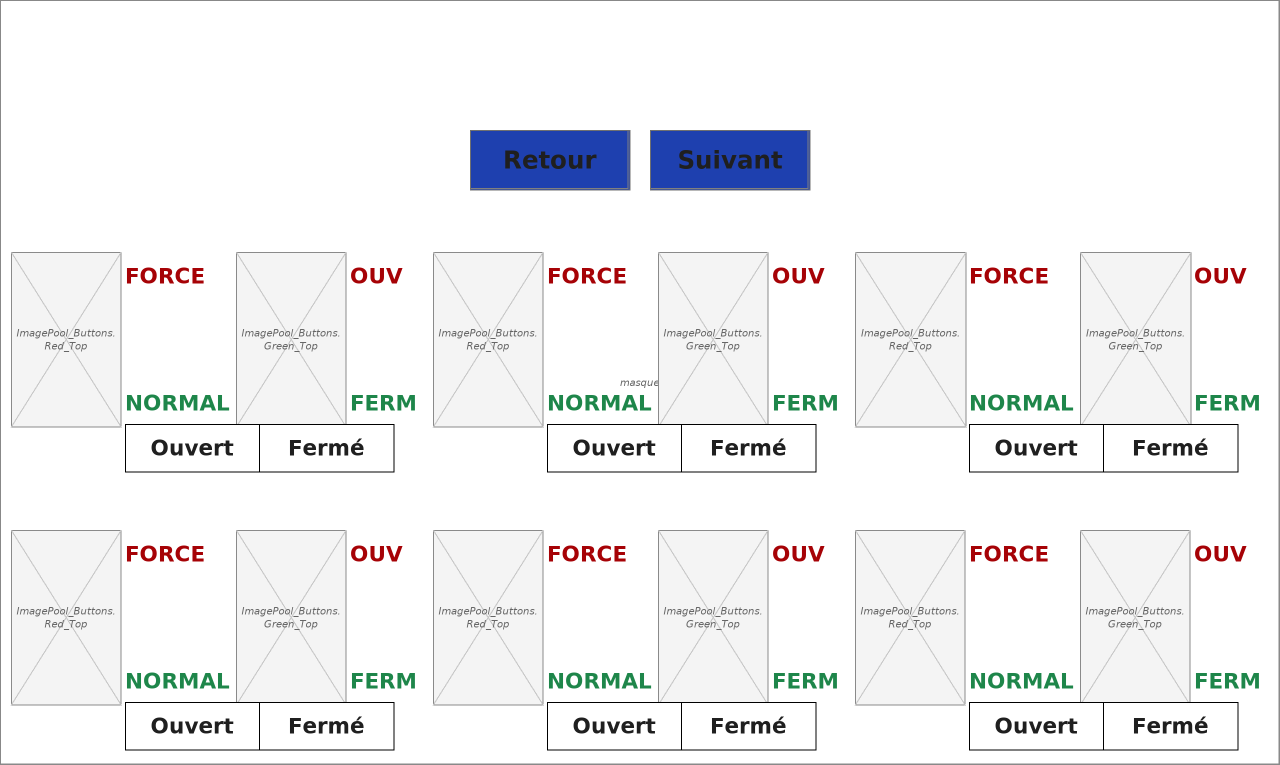
VISUALIZATION Maintenance_2  // 1280x765
    Frame (0,0 1280x765)
        shows masque()
    Button (650,130 160x60), "Suivant"
        OnMouseDown: execute {
            IF (Option_Bas_Debit OR Option_Douchette OR Option_NEP)
            	THEN
            	VisuElems.CURRENTVISU := 'Maintenance_3';
            	ELSIF (Option_WC_GV OR Option_WC_PV OR Option_Prise)
            		THEN
            		VisuElems.CURRENTVISU := 'Maintenance_4';
            	ELSIF (Option_Cabine_Climatique)
            		THEN
            		VisuElems.CURRENTVISU := 'Maintenance_5';
            	ELSIF (Option_Com_RegSouf_Ultrason)
            		THEN
            		VisuElems.CURRENTVISU := 'Maintenance_6';
            	ELSE
            		VisuElems.CURRENTVISU := 'Maintenance_7';
            END_IF
        }
    Button (470,130 160x60), "Retour"
        OnMouseDown: execute {
            IF (Option_RegSouf_Ultrason OR Option_Reg_Etanche_Ext OR Option_V3V_EauMitig)
            	THEN
            	VisuElems.CURRENTVISU := 'Maintenance_1';
            	ELSE
            	VisuElems.CURRENTVISU := 'menu';
            END_IF
        }
    Group (433,212 415x260), invisible if: NOT Option_Douche OR Option_Debitmetre_Douche
        Group (0,40 415x174)
            Group (0,0 225x175)
                Group (0,0 110x175)
                    Image (0,0 110x175), invisible if: EF_Cmd_Vanne_Alim_Douche, image: ImagePool_Buttons.Green_Bottom
                        OnMouseDown: toggle EF_Cmd_Vanne_Alim_Douche
                    Image (0,0 110x175), invisible if: NOT EF_Cmd_Vanne_Alim_Douche, image: ImagePool_Buttons.Red_Top
                        OnMouseDown: toggle EF_Cmd_Vanne_Alim_Douche
                Rectangle (111,0 114x48), "FORCE"
                Rectangle (111,64 114x48), "MODE"
                Rectangle (111,127 114x48), "NORMAL"
            Group (225,0 190x175), invisible if: NOT EF_Cmd_Vanne_Alim_Douche
                Group (0,0 110x175)
                    Image (0,0 110x175), invisible if: F_Cmd_Vanne_Alim_Douche, image: ImagePool_Buttons.Red_Bottom
                        OnMouseDown: toggle F_Cmd_Vanne_Alim_Douche
                    Image (0,0 110x175), invisible if: NOT F_Cmd_Vanne_Alim_Douche, image: ImagePool_Buttons.Green_Top
                        OnMouseDown: toggle F_Cmd_Vanne_Alim_Douche
                Rectangle (111,0 79x48), "OUV"
                Rectangle (111,64 79x48), "OUT"
                Rectangle (111,127 79x48), "FERM"
        Group (33,212 350x48)
            Rectangle (0,0 81x48), "FDC :"
            RoundedRectangle (81,0 135x48), "Ouvert", invisible if: NOT E_Vanne_Alim_Douche_Ouv
            RoundedRectangle (215,0 135x48), "Fermé", invisible if: NOT E_Vanne_Alim_Douche_Ferm
        Rectangle (0,0 415x40), "Vanne douche"
    Group (433,490 415x260), invisible if: NOT Option_Lavabo OR Option_Debitmetre_Lavabo
        Group (0,40 415x174)
            Group (0,0 225x175)
                Group (0,0 110x175)
                    Image (0,0 110x175), invisible if: EF_Cmd_Vanne_Alim_Douche, image: ImagePool_Buttons.Green_Bottom
                        OnMouseDown: toggle EF_Cmd_Vanne_Alim_Douche
                    Image (0,0 110x175), invisible if: NOT EF_Cmd_Vanne_Alim_Douche, image: ImagePool_Buttons.Red_Top
                        OnMouseDown: toggle EF_Cmd_Vanne_Alim_Douche
                Rectangle (111,0 114x48), "FORCE"
                Rectangle (111,64 114x48), "MODE"
                Rectangle (111,127 114x48), "NORMAL"
            Group (225,0 190x175), invisible if: NOT EF_Cmd_Vanne_Alim_Douche
                Group (0,0 110x175)
                    Image (0,0 110x175), invisible if: F_Cmd_Vanne_Alim_Douche, image: ImagePool_Buttons.Red_Bottom
                        OnMouseDown: toggle F_Cmd_Vanne_Alim_Douche
                    Image (0,0 110x175), invisible if: NOT F_Cmd_Vanne_Alim_Douche, image: ImagePool_Buttons.Green_Top
                        OnMouseDown: toggle F_Cmd_Vanne_Alim_Douche
                Rectangle (111,0 79x48), "OUV"
                Rectangle (111,64 79x48), "OUT"
                Rectangle (111,127 79x48), "FERM"
        Group (33,212 350x48)
            Rectangle (0,0 81x48), "FDC :"
            RoundedRectangle (81,0 135x48), "Ouvert", invisible if: NOT E_Vanne_Alim_Lavabo_Ouv
            RoundedRectangle (215,0 135x48), "Fermé", invisible if: NOT E_Vanne_Alim_Lavabo_Ferm
        Rectangle (0,0 415x40), "Vanne lavabo"
    Group (855,212 415x260), invisible if: NOT Option_Douche
        Group (0,40 415x174)
            Group (0,0 225x175)
                Group (0,0 110x175)
                    Image (0,0 111x175), invisible if: EF_Cmd_Vanne_Vid_Douche, image: ImagePool_Buttons.Green_Bottom
                        OnMouseDown: toggle EF_Cmd_Vanne_Vid_Douche
                    Image (0,0 111x175), invisible if: NOT EF_Cmd_Vanne_Vid_Douche, image: ImagePool_Buttons.Red_Top
                        OnMouseDown: toggle EF_Cmd_Vanne_Vid_Douche
                Rectangle (111,0 114x48), "FORCE"
                Rectangle (111,64 114x48), "MODE"
                Rectangle (111,127 114x48), "NORMAL"
            Group (225,0 190x175), invisible if: NOT EF_Cmd_Vanne_Vid_Douche
                Group (0,0 110x175)
                    Image (0,0 111x175), invisible if: F_Cmd_Vanne_Vid_Douche, image: ImagePool_Buttons.Red_Bottom
                        OnMouseDown: toggle F_Cmd_Vanne_Vid_Douche
                    Image (0,0 111x175), invisible if: NOT F_Cmd_Vanne_Vid_Douche, image: ImagePool_Buttons.Green_Top
                        OnMouseDown: toggle F_Cmd_Vanne_Vid_Douche
                Rectangle (111,0 79x48), "OUV"
                Rectangle (111,64 79x48), "OUT"
                Rectangle (111,127 79x48), "FERM"
        Group (33,212 350x48)
            Rectangle (0,0 81x48), "FDC :"
            RoundedRectangle (81,0 135x48), "Ouvert", invisible if: NOT E_Vanne_Vidange_Douche_Ouv
            RoundedRectangle (215,0 135x48), "Fermé", invisible if: NOT E_Vanne_Vidange_Douche_Ferm
        Rectangle (0,0 415x40), "Drain douche"
    Group (855,490 415x260), invisible if: NOT Option_Lavabo
        Group (0,40 415x174)
            Group (0,0 225x175)
                Group (0,0 110x175)
                    Image (0,0 110x175), invisible if: EF_Cmd_Vanne_Vid_Lavabo, image: ImagePool_Buttons.Green_Bottom
                        OnMouseDown: toggle EF_Cmd_Vanne_Vid_Lavabo
                    Image (0,0 110x175), invisible if: NOT EF_Cmd_Vanne_Vid_Lavabo, image: ImagePool_Buttons.Red_Top
                        OnMouseDown: toggle EF_Cmd_Vanne_Vid_Lavabo
                Rectangle (111,0 114x48), "FORCE"
                Rectangle (111,64 114x48), "MODE"
                Rectangle (111,127 114x48), "NORMAL"
            Group (225,0 190x175), invisible if: NOT EF_Cmd_Vanne_Vid_Lavabo
                Group (0,0 110x175)
                    Image (0,0 110x175), invisible if: F_Cmd_Vanne_Vid_Lavabo, image: ImagePool_Buttons.Red_Bottom
                        OnMouseDown: toggle F_Cmd_Vanne_Vid_Lavabo
                    Image (0,0 110x175), invisible if: NOT F_Cmd_Vanne_Vid_Lavabo, image: ImagePool_Buttons.Green_Top
                        OnMouseDown: toggle F_Cmd_Vanne_Vid_Lavabo
                Rectangle (111,0 79x48), "OUV"
                Rectangle (111,64 79x48), "OUT"
                Rectangle (111,127 79x48), "FERM"
        Group (33,212 350x48)
            Rectangle (0,0 81x48), "FDC :"
            RoundedRectangle (81,0 135x48), "Ouvert", invisible if: NOT E_Vanne_Vidange_Lavabo_Ouv
            RoundedRectangle (215,0 135x48), "Fermé", invisible if: NOT E_Vanne_Vidange_Lavabo_Ferm
        Rectangle (0,0 415x40), "Drain lavabo"
    Group (11,212 415x260), invisible if: NOT Option_Douche OR NOT Option_Debitmetre_Douche
        Group (0,40 415x174)
            Group (0,0 225x175)
                Group (0,0 110x175)
                    Image (0,0 110x175), invisible if: EF_Cmd_ElectroValve_Alim_Douche, image: ImagePool_Buttons.Green_Bottom
                    Image (0,0 110x175), invisible if: NOT EF_Cmd_ElectroValve_Alim_Douche, image: ImagePool_Buttons.Red_Top
                Rectangle (111,0 114x48), "FORCE"
                Rectangle (111,64 114x48), "MODE"
                Rectangle (111,127 114x48), "NORMAL"
            Group (225,0 190x175), invisible if: NOT EF_Cmd_ElectroValve_Alim_Douche
                Group (0,0 110x175)
                    Image (0,0 110x175), invisible if: F_Cmd_ElectroValve_Alim_Douche, image: ImagePool_Buttons.Red_Bottom
                        OnMouseDown: toggle F_Cmd_ElectroValve_Alim_Douche
                    Image (0,0 110x175), invisible if: NOT F_Cmd_ElectroValve_Alim_Douche, image: ImagePool_Buttons.Green_Top
                        OnMouseDown: toggle F_Cmd_ElectroValve_Alim_Douche
                Rectangle (111,0 79x48), "OUV"
                Rectangle (111,64 79x48), "OUT"
                Rectangle (111,127 79x48), "FERM"
        Group (33,212 350x48), invisible if: TRUE
            Rectangle (0,0 81x48), "FDC :"
            RoundedRectangle (81,0 135x48), "Ouvert"
            RoundedRectangle (215,0 135x48), "Fermé"
        Rectangle (0,0 415x40), "Electrovanne douche"
    Group (11,490 415x260), invisible if: NOT Option_Lavabo OR NOT Option_Debitmetre_Lavabo
        Group (0,40 415x174)
            Group (0,0 225x175)
                Group (0,0 110x175)
                    Image (0,0 110x175), invisible if: EF_Cmd_ElectroValve_Alim_Lavabo, image: ImagePool_Buttons.Green_Bottom
                        OnMouseDown: toggle EF_Cmd_ElectroValve_Alim_Lavabo
                    Image (0,0 110x175), invisible if: NOT EF_Cmd_ElectroValve_Alim_Lavabo, image: ImagePool_Buttons.Red_Top
                        OnMouseDown: toggle EF_Cmd_ElectroValve_Alim_Lavabo
                Rectangle (111,0 114x48), "FORCE"
                Rectangle (111,64 114x48), "MODE"
                Rectangle (111,127 114x48), "NORMAL"
            Group (225,0 190x175), invisible if: NOT EF_Cmd_ElectroValve_Alim_Lavabo
                Group (0,0 110x175)
                    Image (0,0 110x175), invisible if: F_Cmd_ElectroValve_Alim_Lavabo, image: ImagePool_Buttons.Red_Bottom
                        OnMouseDown: toggle F_Cmd_ElectroValve_Alim_Lavabo
                    Image (0,0 110x175), invisible if: NOT F_Cmd_ElectroValve_Alim_Lavabo, image: ImagePool_Buttons.Green_Top
                        OnMouseDown: toggle F_Cmd_ElectroValve_Alim_Lavabo
                Rectangle (111,0 79x48), "OUV"
                Rectangle (111,64 79x48), "OUT"
                Rectangle (111,127 79x48), "FERM"
        Group (33,212 350x48), invisible if: TRUE
            Rectangle (0,0 81x48), "FDC :"
            RoundedRectangle (81,0 135x48), "Ouvert"
            RoundedRectangle (215,0 135x48), "Fermé"
        Rectangle (0,0 415x40), "Electrovanne lavabo"
END_VISUALIZATION

(* stored: Version 1.1.0.1, ProductVersion 3.1.4024.15
   Visu Maintenance_2: Id {a57c9f42-73a7-4cd2-becb-ce5f505a9bfc} *)
